{attribute 'qualified_only'}
VAR_GLOBAL
	
END_VAR

(* stored: Version 1.1.0.1
   GVL GVL_Test: Id {8909eaec-dbc3-4ff3-b255-cb28f47b4aca} *)
